RoboDK station: segmentscan.rdk

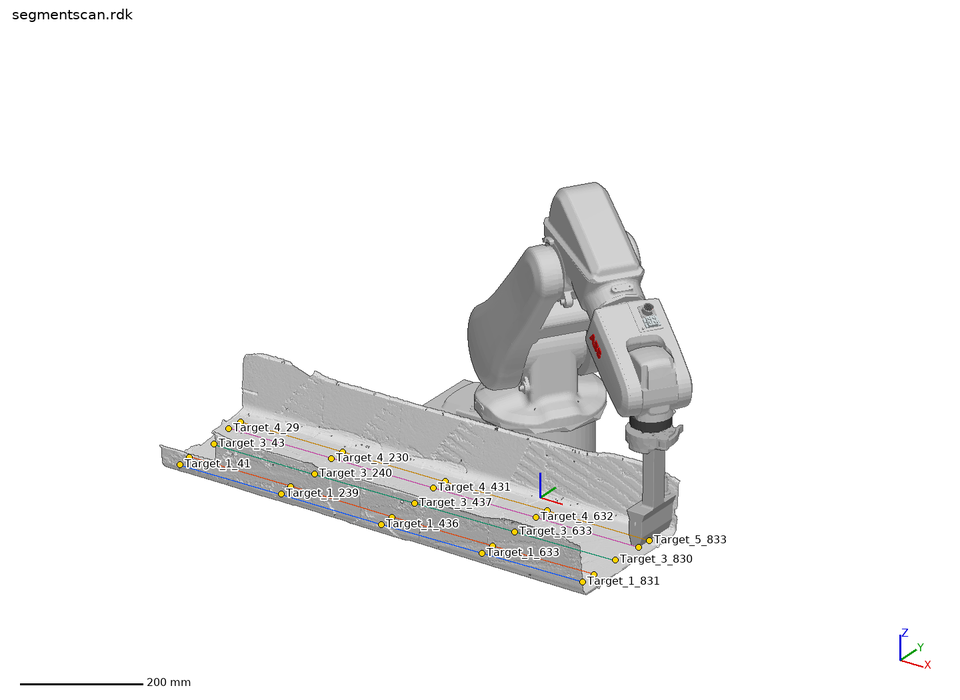
[picture v0: the station drawn from its stored meshes, robots at their saved joint values, targets as dots, program paths as lines]
Station segmentscan (saved by RoboDK 5.6.3). Poses are relative to the parent item; angles as X-Y-Z fixed-axis rotations.
Station parameters (name, value as stored): IO_5, 1, AddPointOnSurface_PointUtilities, 0, AddPointOnSurface_Temp, 1, AddPointOnSurface1_Temp, 1, Updated_Point_on_Surface_Temp, 1, Updated_Point_on_Surface1_Temp, 1, Updated_Point_on_Surface7_Temp, 1
  - frame ABB IRB 120-3/0.6 Base at (0, 0, 0) mm
    - robot ABB IRB 120-3/0.6: 6 axes, payload 3 kg, reach 580 mm, repeatability 0.01 mm, weight 25 kg
        modified DH rows (alpha deg, a mm, theta deg, d mm): 0, 0, 0, 290; -90, 0, -90, 0; 0, 270, 0, 0; -90, 70, 0, 302; 90, 0, 0, 0; -90, 0, 180, 72
        joint limits [-165, -110, -90, -160, -120, -400] to [165, 110, 70, 160, 120, 400]; home [0, 0, 0, 0, 0, 0]; saved at [-32.561, 40.332, -11.466, -0.481, 61.682, 56.527]
      - tool Curved Probe EE Assembly, TCP at (-31.5, 0, 220) mm, size 87.1 x 223.9 x 88.6 mm
      - tool NDI Flat EE, TCP at (0, 0, 205) mm, rotated rx 180 ry 0 rz 90 deg, size 96.8 x 88.5 x 197.8 mm
        - object NDI contour Guide at (0, 0, 0) mm, size 120.9 x 36 x 55.4 mm, geometry from NDI contour Guide.STEP
      - tool curved_frame, TCP at (-30, 0, 220) mm, rotated rx 0 ry 0 rz 90 deg, size 38.2 x 202.5 x 73.3 mm, geometry from curved_frame.stl
    - frame Reference SW at (0, 0, 0) mm
      - object Boeing Test Plate 7 at (0, 0, 0) mm, size 666.8 x 335 x 7 mm, geometry from Boeing Test Plate 7.STL
        - object P[119.10,-424.69,150.00,0.00,0.00,1.00] at (0, 0, 0) mm, 1 curves
        - object P[134.56,-278.64,150.00,0.00,0.00,1.00] at (0, 0, 0) mm, 1 curves
        - object P[-204.50,-248.00,150.00,0.00,0.00,1.00] at (0, 0, 0) mm, 1 curves
        - object P[-165.96,-417.97,150.00,0.00,0.00,1.00] at (0, 0, 0) mm, 1 curves
      - object Spar with Spline at (0, -11, 0) mm, size 840.5 x 321.6 x 114.9 mm, geometry from ABB Table.stl
      - target Target_1_41 (Cartesian target) at (-392.69, -461.66, 133.94) mm, rotated rx -0.59 ry -0.16 rz 1.15 deg; joints [-32.561, 40.332, -11.466, -0.481, 61.682, 56.527] of ABB IRB 120-3/0.6
      - target Target_1_239 (Cartesian target) at (-194.73, -457.7, 134.35) mm, rotated rx -0.59 ry -0.16 rz 1.15 deg; joints [-32.561, 40.332, -11.466, -0.481, 61.682, 56.527] of ABB IRB 120-3/0.6
      - target Target_1_436 (Cartesian target) at (2.24, -453.79, 132.61) mm, rotated rx -0.59 ry -0.16 rz 1.15 deg; joints [-32.561, 40.332, -11.466, -0.481, 61.682, 56.527] of ABB IRB 120-3/0.6
      - target Target_1_633 (Cartesian target) at (199.2, -449.83, 134.44) mm, rotated rx -0.59 ry -0.16 rz 1.15 deg; joints [-32.561, 40.332, -11.466, -0.481, 61.682, 56.527] of ABB IRB 120-3/0.6
      - target Target_1_831 (Cartesian target) at (397.15, -445.86, 136.3) mm, rotated rx -0.59 ry -0.16 rz 1.15 deg; joints [-32.561, 40.332, -11.466, -0.481, 61.682, 56.527] of ABB IRB 120-3/0.6
      - target Target_2_38 (Cartesian target) at (-396.32, -429.89, 133.98) mm, rotated rx -0.59 ry -0.16 rz 1.15 deg; joints [-32.561, 40.332, -11.466, -0.481, 61.682, 56.527] of ABB IRB 120-3/0.6
      - target Target_2_236 (Cartesian target) at (-198.36, -425.93, 134.48) mm, rotated rx -0.59 ry -0.16 rz 1.15 deg; joints [-32.561, 40.332, -11.466, -0.481, 61.682, 56.527] of ABB IRB 120-3/0.6
      - target Target_2_435 (Cartesian target) at (0.6, -421.97, 132.96) mm, rotated rx -0.59 ry -0.16 rz 1.15 deg; joints [-32.561, 40.332, -11.466, -0.481, 61.682, 56.527] of ABB IRB 120-3/0.6
      - target Target_2_633 (Cartesian target) at (198.56, -418.01, 134.39) mm, rotated rx -0.59 ry -0.16 rz 1.15 deg; joints [-32.561, 40.332, -11.466, -0.481, 61.682, 56.527] of ABB IRB 120-3/0.6
      - target Target_2_831 (Cartesian target) at (396.51, -414.03, 136.43) mm, rotated rx -0.59 ry -0.16 rz 1.15 deg; joints [-32.561, 40.332, -11.466, -0.481, 61.682, 56.527] of ABB IRB 120-3/0.6
      - target Target_3_43 (Cartesian target) at (-392.59, -366.14, 132.95) mm, rotated rx -0.61 ry -0.16 rz 1.15 deg; joints [-32.561, 40.332, -11.466, -0.481, 61.682, 56.527] of ABB IRB 120-3/0.6
      - target Target_3_240 (Cartesian target) at (-195.63, -362.22, 131.97) mm, rotated rx -0.59 ry -0.16 rz 1.15 deg; joints [-32.561, 40.332, -11.466, -0.481, 61.682, 56.527] of ABB IRB 120-3/0.6
      - target Target_3_437 (Cartesian target) at (1.33, -358.28, 132.98) mm, rotated rx -0.59 ry -0.16 rz 1.15 deg; joints [-32.561, 40.332, -11.466, -0.481, 61.682, 56.527] of ABB IRB 120-3/0.6
      - target Target_3_633 (Cartesian target) at (197.29, -354.36, 134.16) mm, rotated rx -0.59 ry -0.16 rz 1.15 deg; joints [-32.561, 40.332, -11.466, -0.481, 61.682, 56.527] of ABB IRB 120-3/0.6
      - target Target_3_830 (Cartesian target) at (394.24, -350.4, 136.32) mm, rotated rx -0.59 ry -0.16 rz 1.15 deg; joints [-32.561, 40.332, -11.466, -0.481, 61.682, 56.527] of ABB IRB 120-3/0.6
      - target Target_4_29 (Cartesian target) at (-407.86, -302.78, 131.69) mm, rotated rx -0.59 ry -0.16 rz 1.15 deg; joints [-32.561, 40.332, -11.466, -0.481, 61.682, 56.527] of ABB IRB 120-3/0.6
      - target Target_4_230 (Cartesian target) at (-206.9, -298.77, 131.92) mm, rotated rx -0.59 ry -0.16 rz 1.15 deg; joints [-32.561, 40.332, -11.466, -0.481, 61.682, 56.527] of ABB IRB 120-3/0.6
      - target Target_4_431 (Cartesian target) at (-5.94, -294.75, 132.71) mm, rotated rx -0.59 ry -0.16 rz 1.15 deg; joints [-32.561, 40.332, -11.466, -0.481, 61.682, 56.527] of ABB IRB 120-3/0.6
      - target Target_4_632 (Cartesian target) at (195.02, -290.72, 134.04) mm, rotated rx -0.59 ry -0.16 rz 1.15 deg; joints [-32.561, 40.332, -11.466, -0.481, 61.682, 56.527] of ABB IRB 120-3/0.6
      - target Target_4_833 (Cartesian target) at (395.98, -286.71, 134.24) mm, rotated rx -0.59 ry -0.16 rz 1.15 deg; joints [-32.561, 40.332, -11.466, -0.481, 61.682, 56.527] of ABB IRB 120-3/0.6
      - target Target_5_32 (Cartesian target) at (-405.5, -270.89, 131.86) mm, rotated rx -0.59 ry -0.16 rz 1.15 deg; joints [-32.561, 40.332, -11.466, -0.481, 61.682, 56.527] of ABB IRB 120-3/0.6
      - target Target_5_232 (Cartesian target) at (-205.54, -266.9, 132.05) mm, rotated rx -0.59 ry -0.16 rz 1.15 deg; joints [-32.561, 40.332, -11.466, -0.481, 61.682, 56.527] of ABB IRB 120-3/0.6
      - target Target_5_433 (Cartesian target) at (-4.58, -262.88, 132.78) mm, rotated rx -0.59 ry -0.16 rz 1.15 deg; joints [-32.561, 40.332, -11.466, -0.481, 61.682, 56.527] of ABB IRB 120-3/0.6
      - target Target_5_633 (Cartesian target) at (195.38, -258.87, 134.09) mm, rotated rx -0.59 ry -0.16 rz 1.15 deg; joints [-32.561, 40.332, -11.466, -0.481, 61.682, 56.527] of ABB IRB 120-3/0.6
      - target Target_5_833 (Cartesian target) at (395.34, -254.88, 134.35) mm, rotated rx -0.59 ry -0.16 rz 1.15 deg; joints [-32.561, 40.332, -11.466, -0.481, 61.682, 56.527] of ABB IRB 120-3/0.6
  - Python program Updated Point on Surface (listed below)
  - object Flat Plate Curve at (0, 0, 0) mm, geometry from  V 25.
  - object scan3_test_cleaned at (0, 0, 0) mm, size 856.2 x 311 x 115.1 mm, geometry from scan3_test_cleaned.ply
  - program Path_1 (5 instructions, listed below)
  - program Path_2 (5 instructions, listed below)
  - program Path_3 (5 instructions, listed below)
  - program Path_4 (5 instructions, listed below)
  - program Path_5 (5 instructions, listed below)
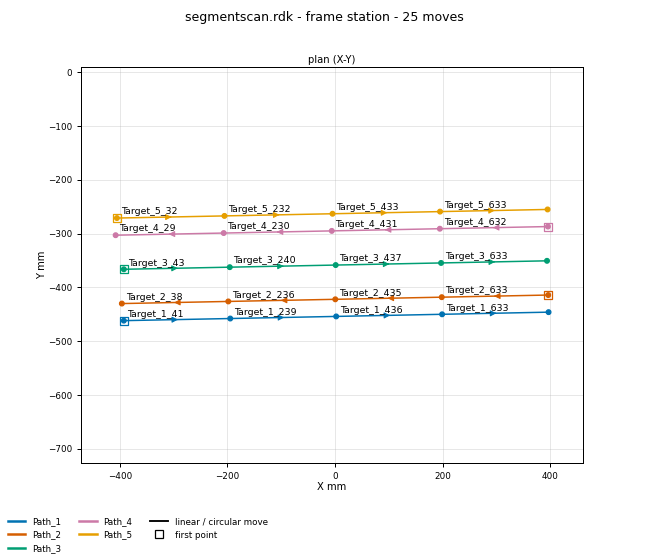
[picture p0: tool path of segmentscan.rdk in frame station, 25 of 25 moves have a stored position in this frame; points joined in program order, loops and branches not executed]

--- Python program Updated Point on Surface ---
# --------------------------------------------
# This Code combines Atsushi Sakai's Grid Based Sweeping
# and RoboDK's AddPointOnSurface to generate a raster path
# on a FLAT surface.

# Python Robotics - GridBased Sweeping: https://github.com/AtsushiSakai/PythonRobotics/tree/master
# RoboDK's - AddPointToSurface: https://github.com/RoboDK/Plug-In-Interface/tree/master
#-----------------------------------------------

#

from robodk import robolink, roboapps, robodialogs, robomath
RDK = robolink.Robolink()

from PointUtilities import Settings

import math
from enum import IntEnum
import numpy as np
import matplotlib.pyplot as plt
import sys
import pathlib
sys.path.append(str(pathlib.Path(__file__).parent.parent.parent))

from utils.angle import rot_mat_2d
from Mapping.grid_map_lib.grid_map_lib import GridMap, FloatGrid

class SweepSearcher:
    class SweepDirection(IntEnum):
        UP = 1
        DOWN = -1

    class MovingDirection(IntEnum):
        RIGHT = 1
        LEFT = -1

    def __init__(self,
                 moving_direction, sweep_direction, x_inds_goal_y, goal_y):
        self.moving_direction = moving_direction
        self.sweep_direction = sweep_direction
        self.turing_window = []
        self.update_turning_window()
        self.x_indexes_goal_y = x_inds_goal_y
        self.goal_y = goal_y

    def move_target_grid(self, c_x_index, c_y_index, grid_map):
        n_x_index = self.moving_direction + c_x_index
        n_y_index = c_y_index

        # found safe grid
        if not self.check_occupied(n_x_index, n_y_index, grid_map):
            return n_x_index, n_y_index
        else:  # occupied
            next_c_x_index, next_c_y_index = self.find_safe_turning_grid(
                c_x_index, c_y_index, grid_map)
            if (next_c_x_index is None) and (next_c_y_index is None):
                # moving backward
                next_c_x_index = -self.moving_direction + c_x_index
                next_c_y_index = c_y_index
                if self.check_occupied(next_c_x_index, next_c_y_index, grid_map):
                    # moved backward, but the grid is occupied by obstacle
                    return None, None
            else:
                # keep moving until end
                while not self.check_occupied(next_c_x_index + self.moving_direction, next_c_y_index, grid_map):
                    next_c_x_index += self.moving_direction
                self.swap_moving_direction()
            return next_c_x_index, next_c_y_index

    @staticmethod
    def check_occupied(c_x_index, c_y_index, grid_map):
        return grid_map.check_occupied_from_xy_index(c_x_index, c_y_index, FloatGrid(0.5))

    def find_safe_turning_grid(self, c_x_index, c_y_index, grid_map):

        for (d_x_ind, d_y_ind) in self.turing_window:

            next_x_ind = d_x_ind + c_x_index
            next_y_ind = d_y_ind + c_y_index

            # found safe grid
            if not self.check_occupied(next_x_ind, next_y_ind, grid_map):
                return next_x_ind, next_y_ind

        return None, None

    def is_search_done(self, grid_map):
        for ix in self.x_indexes_goal_y:
            if not self.check_occupied(ix, self.goal_y, grid_map):
                return False

        # all lower grid is occupied
        return True

    def update_turning_window(self):
        # turning window definition
        # robot can move grid based on it.
        self.turing_window = [
            (self.moving_direction, 0.0),
            (self.moving_direction, self.sweep_direction),
            (0, self.sweep_direction),
            (-self.moving_direction, self.sweep_direction),
        ]

    def swap_moving_direction(self):
        self.moving_direction *= -1
        self.update_turning_window()

    def search_start_grid(self, grid_map):
        x_inds = []
        y_ind = 0
        if self.sweep_direction == self.SweepDirection.DOWN:
            x_inds, y_ind = search_free_grid_index_at_edge_y(
                grid_map, from_upper=True)
        elif self.sweep_direction == self.SweepDirection.UP:
            x_inds, y_ind = search_free_grid_index_at_edge_y(
                grid_map, from_upper=False)

        if self.moving_direction == self.MovingDirection.RIGHT:
            return min(x_inds), y_ind
        elif self.moving_direction == self.MovingDirection.LEFT:
            return max(x_inds), y_ind

        raise ValueError("self.moving direction is invalid ")


def find_sweep_direction_and_start_position(ox, oy):
    # find sweep_direction
    max_dist = 0.0
    vec = [0.0, 0.0]
    sweep_start_pos = [0.0, 0.0]
    for i in range(len(ox) - 1):
        dx = ox[i + 1] - ox[i]
        dy = oy[i + 1] - oy[i]
        d = np.hypot(dx, dy)

        if d > max_dist:
            max_dist = d
            vec = [dx, dy]
            sweep_start_pos = [ox[i], oy[i]]

    return vec, sweep_start_pos


def convert_grid_coordinate(ox, oy, sweep_vec, sweep_start_position):
    tx = [ix - sweep_start_position[0] for ix in ox]
    ty = [iy - sweep_start_position[1] for iy in oy]
    th = math.atan2(sweep_vec[1], sweep_vec[0])
    converted_xy = np.stack([tx, ty]).T @ rot_mat_2d(th)

    return converted_xy[:, 0], converted_xy[:, 1]


def convert_global_coordinate(x, y, sweep_vec, sweep_start_position):
    th = math.atan2(sweep_vec[1], sweep_vec[0])
    converted_xy = np.stack([x, y]).T @ rot_mat_2d(-th)
    rx = [ix + sweep_start_position[0] for ix in converted_xy[:, 0]]
    ry = [iy + sweep_start_position[1] for iy in converted_xy[:, 1]]
    return rx, ry


def search_free_grid_index_at_edge_y(grid_map, from_upper=False):
    y_index = None
    x_indexes = []

    if from_upper:
        x_range = range(grid_map.height)[::-1]
        y_range = range(grid_map.width)[::-1]
    else:
        x_range = range(grid_map.height)
        y_range = range(grid_map.width)

    for iy in x_range:
        for ix in y_range:
            if not SweepSearcher.check_occupied(ix, iy, grid_map):
                y_index = iy
                x_indexes.append(ix)
        if y_index:
            break

    return x_indexes, y_index


def setup_grid_map(ox, oy, resolution, sweep_direction, offset_grid=10):
    width = math.ceil((max(ox) - min(ox)) / resolution) + offset_grid
    height = math.ceil((max(oy) - min(oy)) / resolution) + offset_grid
    center_x = (np.max(ox) + np.min(ox)) / 2.0
    center_y = (np.max(oy) + np.min(oy)) / 2.0

    grid_map = GridMap(width, height, resolution, center_x, center_y)
    grid_map.print_grid_map_info()
    grid_map.set_value_from_polygon(ox, oy, FloatGrid(1.0), inside=False)
    grid_map.expand_grid()

    x_inds_goal_y = []
    goal_y = 0
    if sweep_direction == SweepSearcher.SweepDirection.UP:
        x_inds_goal_y, goal_y = search_free_grid_index_at_edge_y(
            grid_map, from_upper=True)
    elif sweep_direction == SweepSearcher.SweepDirection.DOWN:
        x_inds_goal_y, goal_y = search_free_grid_index_at_edge_y(
            grid_map, from_upper=False)

    return grid_map, x_inds_goal_y, goal_y


def sweep_path_search(sweep_searcher, grid_map, grid_search_animation=False):
    # search start grid
    c_x_index, c_y_index = sweep_searcher.search_start_grid(grid_map)
    if not grid_map.set_value_from_xy_index(c_x_index, c_y_index, FloatGrid(0.5)):
        print("Cannot find start grid")
        return [], []

    x, y = grid_map.calc_grid_central_xy_position_from_xy_index(c_x_index,
                                                                c_y_index)
    px, py = [x], [y]

    fig, ax = None, None
    if grid_search_animation:
        fig, ax = plt.subplots()
        # for stopping simulation with the esc key.
        fig.canvas.mpl_connect(
            'key_release_event',
            lambda event: [exit(0) if event.key == 'escape' else None])

    while True:
        c_x_index, c_y_index = sweep_searcher.move_target_grid(c_x_index,
                                                               c_y_index,
                                                               grid_map)

        if sweep_searcher.is_search_done(grid_map) or (
                c_x_index is None or c_y_index is None):
            print("Done")
            break

        x, y = grid_map.calc_grid_central_xy_position_from_xy_index(
            c_x_index, c_y_index)

        px.append(x)
        py.append(y)

        grid_map.set_value_from_xy_index(c_x_index, c_y_index, FloatGrid(0.5))

        if grid_search_animation:
            grid_map.plot_grid_map(ax=ax)
            plt.pause(.5)

    return px, py


def planning(ox, oy, resolution,
             moving_direction=SweepSearcher.MovingDirection.RIGHT,
             sweeping_direction=SweepSearcher.SweepDirection.UP,
             ):
    sweep_vec, sweep_start_position = find_sweep_direction_and_start_position(
        ox, oy)

    rox, roy = convert_grid_coordinate(ox, oy, sweep_vec,
                                       sweep_start_position)

    grid_map, x_inds_goal_y, goal_y = setup_grid_map(rox, roy, resolution,
                                                     sweeping_direction)

    sweep_searcher = SweepSearcher(moving_direction, sweeping_direction,
                                   x_inds_goal_y, goal_y)

    px, py = sweep_path_search(sweep_searcher, grid_map)

    rx, ry = convert_global_coordinate(px, py, sweep_vec,
                                       sweep_start_position)

    print("Path length:", len(rx))

    return rx, ry


# Point Selection
#---------------------------------------

def AddPointOnSurface(RDK=None, S=None):
    """
    Click an object's surface to add a point at that location.
    Points can be added as long as this action is running.
    """
    points = robodialogs.InputDialog('How many Points Would You Like to Select? \n\nEnter an integer:', 0)
    if points <= 0:
        roboapps.Exit()
    else:
        print('Number of Points Selected:', points)

    A = []


    point_counter = 0

    if RDK is None:
        RDK = robolink.Robolink()

    if S is None:
        S = Settings.Settings()
        S.Load(RDK)

    # Clear the selection so that we get a 'rising edge'
    RDK.setSelection([])

    APP = roboapps.RunApplication()
    while APP.Run():

        # Get the point under the mouse
        selected_object, feature_type, _, _, _ = RDK.GetPoints(robolink.FEATURE_HOVER_OBJECT)
        if feature_type != robolink.FEATURE_SURFACE or not selected_object.Valid() or selected_object.Type() not in [robolink.ITEM_TYPE_OBJECT]:
            continue

        # Capture user-click
        if selected_object in RDK.Selection():

            # Get the mouse point on surface
            point_mouse, _ = selected_object.GetPoints(robolink.FEATURE_SURFACE)
            if not point_mouse:
                continue

            # Clear the selection so that we get a 'rising edge'
            RDK.setSelection([])

            # Get the mouse position and normal
            xyzijk = point_mouse[0][0:6]
            xyz = xyzijk[0:3]
            ijk = xyzijk[3:6]

            # Get the mouse position on the surface of the object
            pose_offset = selected_object.Pose()
            xyz_offset = pose_offset * xyz
            ijk_offset = pose_offset[0:3, 0:3] * ijk
            xyzijk = xyz_offset + ijk_offset


            # Add the point to the clicked object, or create a new object
            point_object = selected_object.AddPoints([xyzijk], S.ADD_TO_OBJECT, robolink.PROJECTION_ALONG_NORMAL_RECALC)
            if not S.ADD_TO_OBJECT:
                x, y, z, i, j, k = xyzijk
                point_object.setName(f"P[{x:.2f},{y:.2f},{z:.2f},{i:.2f},{j:.2f},{k:.2f}]")
                point_counter += 1
                A.append(xyzijk)
                print("Point Counter:", point_counter)
                print(A)


                if point_counter >= points:
                    #roboapps.Exit()
                    Check = robodialogs.ShowMessageYesNo('These Points Correct', title=None)
                    if Check == True:
                        resolution = robodialogs.InputDialog('How much overlap (mm)\n\nEnter an integer:', 0)

                        x_coord=[point[0] for point in A]
                        y_coord=[point[1] for point in A]
                        z_coord=[point[2] for point in A]

                        x_coord.append(x_coord[0])
                        y_coord.append(y_coord[0])
                        z_coord.append(z_coord[0])

                        print(x_coord)
                        print(y_coord)


                        px, py = planning(x_coord, y_coord, resolution)
                        pz = len(px)*[sum(z_coord)/len(z_coord)]



                        raster = robomath.Mat([px,py,pz])
                        Raster = RDK.AddCurve(raster)

                        roboapps.Exit()

##                    else:
##                        list_names = RDK.ItemList()  # list all names
##                        for item_name in list_names:
##                            if item_name.startswith('Auto'):
##                                RDK.Item(item_name).Delete()




#---------------------------------------


def runmain():


    if roboapps.Unchecked():
        roboapps.Exit()
    else:
        AddPointOnSurface()



if __name__ == '__main__':
    runmain()

--- program Path_1 (robot ABB IRB 120-3/0.6) ---
  MoveL (Target_1_41)
  MoveL (Target_1_239)
  MoveL (Target_1_436)
  MoveL (Target_1_633)
  MoveL (Target_1_831)

--- program Path_2 (robot ABB IRB 120-3/0.6) ---
  MoveL (Target_2_831)
  MoveL (Target_2_633)
  MoveL (Target_2_435)
  MoveL (Target_2_236)
  MoveL (Target_2_38)

--- program Path_3 (robot ABB IRB 120-3/0.6) ---
  MoveL (Target_3_43)
  MoveL (Target_3_240)
  MoveL (Target_3_437)
  MoveL (Target_3_633)
  MoveL (Target_3_830)

--- program Path_4 (robot ABB IRB 120-3/0.6) ---
  MoveL (Target_4_833)
  MoveL (Target_4_632)
  MoveL (Target_4_431)
  MoveL (Target_4_230)
  MoveL (Target_4_29)

--- program Path_5 (robot ABB IRB 120-3/0.6) ---
  MoveL (Target_5_32)
  MoveL (Target_5_232)
  MoveL (Target_5_433)
  MoveL (Target_5_633)
  MoveL (Target_5_833)
